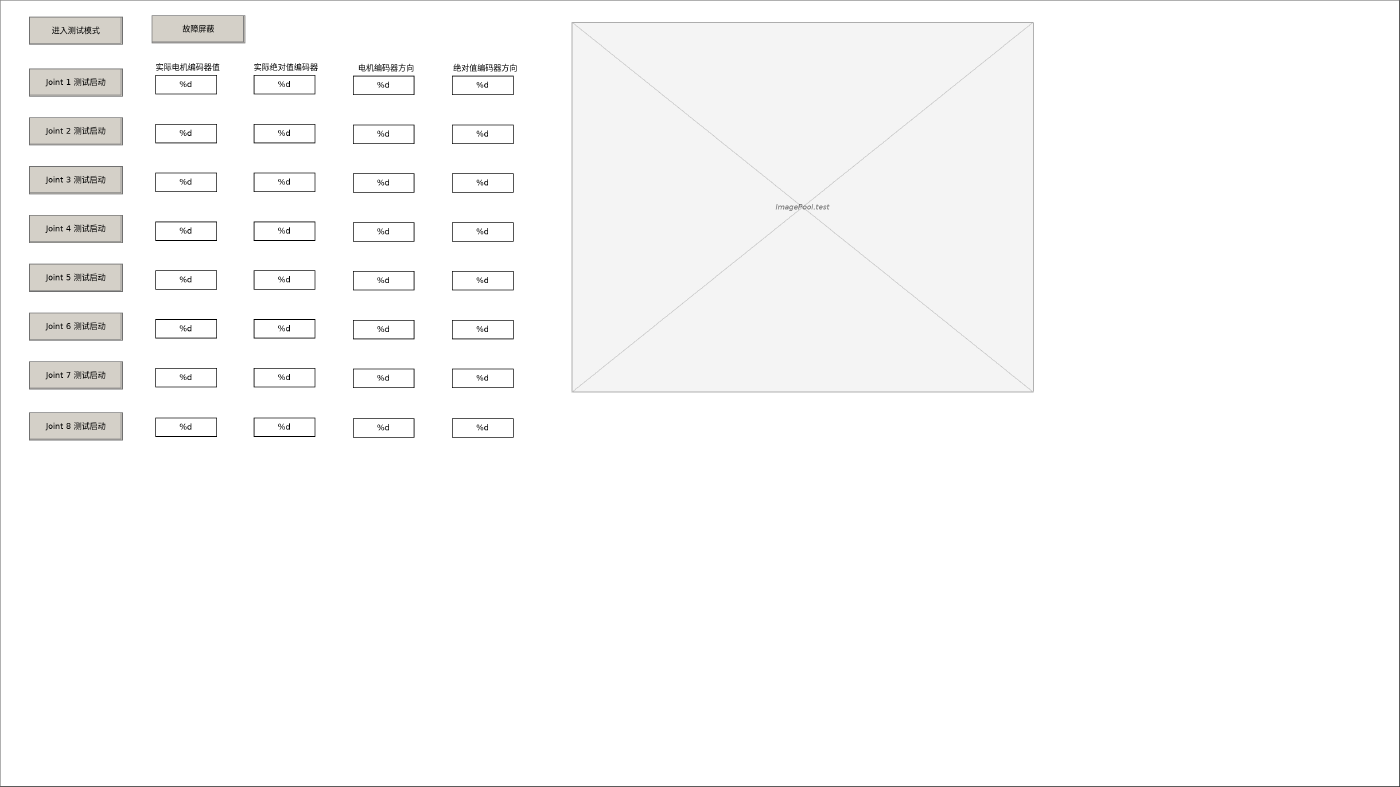
VISUALIZATION arm1JointDir  // 1920x1080
    Rectangle (0,0 1920x1080)
    Image (784,30 633x508), image: ImagePool.test
    Button (40,496 128x38), "Joint 7 测试启动", colour toggle: GVL_armCali.g_jointIntoCaliState[1][7]
        toggle GVL_armCali.g_jointIntoCaliState[1][7]
    Button (40,23 128x38), "进入测试模式", colour toggle: GVL_armCali.g_armEnterCaliMode[1]
        toggle GVL_armCali.g_armEnterCaliMode[1]
    Button (40,94 128x38), "Joint 1 测试启动", colour toggle: GVL_armCali.g_jointIntoCaliState[1][1]
        toggle GVL_armCali.g_jointIntoCaliState[1][1]
    Button (40,161 128x38), "Joint 2 测试启动", colour toggle: GVL_armCali.g_jointIntoCaliState[1][2]
        toggle GVL_armCali.g_jointIntoCaliState[1][2]
    Button (40,228 128x38), "Joint 3 测试启动", colour toggle: GVL_armCali.g_jointIntoCaliState[1][3]
        toggle GVL_armCali.g_jointIntoCaliState[1][3]
    Button (40,295 128x38), "Joint 4 测试启动", colour toggle: GVL_armCali.g_jointIntoCaliState[1][4]
        toggle GVL_armCali.g_jointIntoCaliState[1][4]
    Button (40,362 128x38), "Joint 5 测试启动", colour toggle: GVL_armCali.g_jointIntoCaliState[1][5]
        toggle GVL_armCali.g_jointIntoCaliState[1][5]
    Button (40,429 128x38), "Joint 6 测试启动", colour toggle: GVL_armCali.g_jointIntoCaliState[1][6]
        toggle GVL_armCali.g_jointIntoCaliState[1][6]
    Button (40,566 128x38), "Joint 8 测试启动", colour toggle: GVL_armCali.g_jointIntoCaliState[1][8]
        toggle GVL_armCali.g_jointIntoCaliState[1][8]
    Rectangle (213,103 84x26), "%d", text variable: SetupArmControl.m_setupRobot.m_setupArms[1].m_joints[1].m_motorInputs.m_motorEncoder
    Label (200,81 115x23), "实际电机编码器值"
    Rectangle (348,103 84x26), "%d", text variable: SetupArmControl.m_setupRobot.m_setupArms[1].m_joints[1].m_motorInputs.m_linkEncoder
    Label (335,81 114x23), "实际绝对值编码器"
    Rectangle (213,170 84x26), "%d", text variable: SetupArmControl.m_setupRobot.m_setupArms[1].m_joints[2].m_motorInputs.m_motorEncoder
    Rectangle (348,170 84x26), "%d", text variable: SetupArmControl.m_setupRobot.m_setupArms[1].m_joints[2].m_motorInputs.m_linkEncoder
    Rectangle (213,237 84x26), "%d", text variable: SetupArmControl.m_setupRobot.m_setupArms[1].m_joints[3].m_motorInputs.m_motorEncoder
    Rectangle (348,237 84x26), "%d", text variable: SetupArmControl.m_setupRobot.m_setupArms[1].m_joints[3].m_motorInputs.m_linkEncoder
    Rectangle (213,304 84x26), "%d", text variable: SetupArmControl.m_setupRobot.m_setupArms[1].m_joints[4].m_motorInputs.m_motorEncoder
    Rectangle (348,304 84x26), "%d", text variable: SetupArmControl.m_setupRobot.m_setupArms[1].m_joints[4].m_motorInputs.m_linkEncoder
    Rectangle (213,371 84x26), "%d", text variable: SetupArmControl.m_setupRobot.m_setupArms[1].m_joints[5].m_motorInputs.m_motorEncoder
    Rectangle (348,371 84x26), "%d", text variable: SetupArmControl.m_setupRobot.m_setupArms[1].m_joints[5].m_motorInputs.m_linkEncoder
    Rectangle (213,438 84x26), "%d", text variable: SlaveArmControl.m_slaveRobot.m_slaveArms[1].m_joints[1].m_motorInputs.m_motorEncoder
    Rectangle (348,438 84x26), "%d", text variable: SlaveArmControl.m_slaveRobot.m_slaveArms[1].m_joints[1].m_motorInputs.m_linkEncoder
    Rectangle (213,505 84x26), "%d", text variable: SlaveArmControl.m_slaveRobot.m_slaveArms[1].m_joints[2].m_motorInputs.m_motorEncoder
    Rectangle (348,505 84x26), "%d", text variable: SlaveArmControl.m_slaveRobot.m_slaveArms[1].m_joints[2].m_motorInputs.m_linkEncoder
    Rectangle (213,573 84x26), "%d", text variable: SlaveArmControl.m_slaveRobot.m_slaveArms[1].m_joints[3].m_motorInputs.m_motorEncoder
    Rectangle (348,573 84x26), "%d", text variable: SlaveArmControl.m_slaveRobot.m_slaveArms[1].m_joints[3].m_motorInputs.m_linkEncoder
    Rectangle (484,104 84x26), "%d", text variable: GVL_SetupMotorParameters.g_motorDir[1]
    Label (471,82 117x23), "电机编码器方向"
    Rectangle (484,171 84x26), "%d", text variable: GVL_SetupMotorParameters.g_motorDir[2]
    Rectangle (484,238 84x26), "%d", text variable: GVL_SetupMotorParameters.g_motorDir[3]
    Rectangle (484,305 84x26), "%d", text variable: GVL_SetupMotorParameters.g_motorDir[4]
    Rectangle (484,372 84x26), "%d", text variable: GVL_SetupMotorParameters.g_motorDir[5]
    Rectangle (484,439 84x26), "%d", text variable: GVL_SlaveMotorParameters.g_motorDir[1]
    Rectangle (484,506 84x26), "%d", text variable: GVL_SlaveMotorParameters.g_motorDir[2]
    Rectangle (484,574 84x26), "%d", text variable: GVL_SlaveMotorParameters.g_motorDir[3]
    Rectangle (620,104 84x26), "%d", text variable: GVL_SetupJointEncoderCaliData.g_asbEncoderDir[1]
    Label (607,82 117x23), "绝对值编码器方向"
    Rectangle (620,171 84x26), "%d", text variable: GVL_SetupJointEncoderCaliData.g_asbEncoderDir[2]
    Rectangle (620,238 84x26), "%d", text variable: GVL_SetupJointEncoderCaliData.g_asbEncoderDir[3]
    Rectangle (620,305 84x26), "%d", text variable: GVL_SetupJointEncoderCaliData.g_asbEncoderDir[4]
    Rectangle (620,372 84x26), "%d", text variable: GVL_SetupJointEncoderCaliData.g_asbEncoderDir[5]
    Rectangle (620,439 84x26), "%d", text variable: GVL_SlaveJointEncoderCaliData.g_asbEncoderDir[1]
    Rectangle (620,506 84x26), "%d", text variable: GVL_SlaveJointEncoderCaliData.g_asbEncoderDir[2]
    Rectangle (620,574 84x26), "%d", text variable: GVL_SlaveJointEncoderCaliData.g_asbEncoderDir[3]
    Button (208,21 128x38), "故障屏蔽", colour toggle: g_specialSignal.m_faultMask[1]
        toggle g_specialSignal.m_faultMask[1]
END_VISUALIZATION

(* stored: Version 1.1.0.1, ProductVersion 3.1.4024.11
   Visu arm1JointDir: Id {49ea7e46-c232-42d4-a49b-84494d20e462} *)
